(* IEC 61131-3 sources: SimaticAX/src, 3 files *)

(* ---- basicmotor.st ---- *)
NAMESPACE Motors
    CLASS BasicMotor
        VAR
            status : BOOL;
        END_VAR

        METHOD PUBLIC Start : BOOL
            status := TRUE;
        END_METHOD

        METHOD PUBLIC Stop : BOOL
            status := FALSE;
        END_METHOD

        METHOD PUBLIC IsRunning : BOOL
            isRunning := status;
        END_METHOD
    END_CLASS

END_NAMESPACE

(* ---- configuration.st ---- *)
CONFIGURATION MyConfiguration
    TASK Main(Priority := 1);

    PROGRAM P1 WITH Main: MainProgram;

    VAR_GLOBAL
        startmotor: BOOL;
        stopmotor: BOOL;
    END_VAR
END_CONFIGURATION

(* ---- MainProgram.st ---- *)
USING Motors;

PROGRAM MainProgram
    VAR_EXTERNAL
        startmotor: BOOL;
        stopmotor: BOOL;
    END_VAR

    VAR
        motorA : BasicMotor;
    END_VAR

    IF startmotor THEN
        motorA.Start();
    END_IF;

END_PROGRAM
